// TwinCAT 3 PLC project PLCproj
// ProgramVersion: 3.1.4020.10
// libraries:
//   Tc2_Database, * (Beckhoff Automation GmbH)
//   Tc2_Standard, * (Beckhoff Automation GmbH)
//   Tc2_System, * (Beckhoff Automation GmbH)
//   Tc2_Utilities, * (Beckhoff Automation GmbH)
//   Tc3_Module, * (Beckhoff Automation GmbH)
//   VisuDialogs, * (System)
// project tree:
//   DUTs/ E_ACtype.TcDUT, E_Direction.TcDUT, E_Nchannel.TcDUT, ST_Terminal.TcDUT
//   / GlobalTextList.TcGTLO, PlcTask.TcTTO, Visualization Manager.TcVMO (not stored)
//   GVLs/ GVL.TcGVL, GVL_Checks.TcGVL
//   POUs/ FB_WriteReportToFile.TcPOU, F_Scaling.TcPOU, MAIN.TcPOU, P_Test.TcPOU
//   POUs/Checks/ CheckBounds.TcPOU, CheckDivDInt.TcPOU, CheckDivLInt.TcPOU, CheckDivLReal.TcPOU, CheckDivReal.TcPOU, CheckPointer.TcPOU, CheckRangeSigned.TcPOU, CheckRangeUnsigned.TcPOU
//   VISUs/ Screen1.TcVIS, Obrazki.TcIPO (not stored)
//   VISUs/TextList/ TL_ACtype.TcTLO, TL_BitConventer.TcTLO, TL_Busy.TcTLO, TL_Device.TcTLO, TL_Direction.TcTLO, TL_Nchannel.TcTLO
// real-time tasks:
//   TASK PlcTask: cycle T#10ms, priority 20, ADS port 350
// I/O:
//   DEVICE Device 2 (CX-BK)
//     Box 1 (CX-BK)
// variable links:
//   PLCproj/PLCproj Instance <-> Device 2 (CX-BK)/Box 1 (CX-BK)
//     PlcTask Inputs/GVL.aiINchannel[{1..4}] <-> Term 3 (KL3064)/Channel {1..4}/Data In  (4 links)
//     PlcTask Outputs/GVL.aiOUTchannel[{1..4}] <-> Term 2 (KL4404)/Channel {1..4}/Data Out  (4 links)

CONFIGURATION PLCproj
    RESOURCE PLC ON TwinCAT3
        TASK PlcTask(INTERVAL := T#10ms, PRIORITY := 20);
        PROGRAM MAIN WITH PlcTask : MAIN;
    END_RESOURCE
END_CONFIGURATION

// ---- DUTs/E_ACtype.TcDUT
TYPE E_ACtype :
(
	eACtype_null		:= 0,
	eACtype_0_10V		:= 1,
	eACtype_pl_min10V	:= 2,
	eACtype_0_20mA	:= 3,
	eACtype_4_20mA	:= 4
);
END_TYPE

// ---- DUTs/E_Direction.TcDUT
TYPE E_Direction :
(
	eDirection_null := 0,
	eDirection_Input_Module := 1,
	eDirection_Output_Module := 2
);
END_TYPE

// ---- DUTs/E_Nchannel.TcDUT
TYPE E_Nchannel :
(
	eNchannel_null := 0,
	eNchannel_2 := 1,
	eNchannel_4 := 2,
	eNchannel_8 := 3
);
END_TYPE

// ---- DUTs/ST_Terminal.TcDUT
TYPE ST_Terminal :
STRUCT
	usiDirection		:	USINT;							// Input=1  Output=2
	usiACtype			:	USINT;							// 0..10__±10V__0..20mA__4..20mA 
	usiNchannel			:	USINT;							// Amount of channel
	usiBitConventer		:	USINT;							// N-bit conventer
	sParameters			:	STRING(256);					// Message displayed in HMI during setup terminal type
END_STRUCT
END_TYPE

// ---- GVLs/GVL.TcGVL
VAR_GLOBAL
	 aiINchannel		AT %I*	:	ARRAY [1..8] OF  INT;
	 aiOUTchannel		AT %Q*	:	ARRAY [1..8] OF  INT;
	 

	 
	// aiINchannel		:	ARRAY [1..8] OF  INT;
	// aiOUTchannel		:	ARRAY [1..8] OF  INT;
END_VAR

// ---- GVLs/GVL_Checks.TcGVL
{attribute 'qualified_only'}
VAR_GLOBAL PERSISTENT
	dCheckBounds		: DINT;	(*Licznik przekroczen zakresu indexow, np. tablic*)
	dCheckDivDInt		: DINT;	(*Licznik prob dzielenia Dint przez 0*)
	dCheckDivLInt		: DINT; (*Licznik prob dzielenia LInt przez 0*)
	dCheckDivLReal		: DINT; (*Licznik prob dzielenia LREAL przez 0*)
	dCheckDivReal		: DINT; (*Licznik prob dzielenia REAL przez 0*)
	dCheckRangeSigned	: DINT;	(*Licznik przekroczen  liczby znakowej*)
	dCheckRangeUnsigned	: DINT; (*Licznik przekroczen  liczby bezznakowej*)
END_VAR

// ---- POUs/MAIN.TcPOU
(************************************************************************************)
(*							Beckhoff Automation Poland								*)
(*									13.09.2016										*)
(*								autor: Piotr Szyszka								*)
(*		Analog tester. Allows to chceck suspected with referenced terminal.			*)
(*						Please check preferences in local files.					*)
(*__________________________________________________________________________________*)
PROGRAM MAIN
VAR

END_VAR

P_Test();

END_PROGRAM

// ---- POUs/P_Test.TcPOU
(************************************************************************************)
(*							Beckhoff Automation Poland								*)
(*									13.09.2016										*)
(*								Analog terminal tester								*)
(*								autor: Piotr Szyszka								*)
(*																					*)
(*__________________________________________________________________________________*)
PROGRAM P_Test
VAR
// Choose bus terminals
bReadData			:	BOOL;							// Read Structure
bErrorReadData		:	BOOL;							// Setted not all parametres
bDataSend			:	BOOL;							// Data aquired
stRefTerminal		:	ST_Terminal;
stTestTerminal		:	ST_Terminal;
rtReadData			:	R_TRIG;
ftClearComboBox		:	F_TRIG;
sStatusBox			:	STRING(255)		:='Idle';
sBuffer				:	STRING(255);

eDirection1			:	E_Direction;					// Input=1  Output=2
eDirection2			:	E_Direction;
eACtype				:	E_ACtype;						// 0..10V=1	±10V=2	0..20mA=3	4..20mA=4
eNchannel			:	E_Nchannel;						// 2channels=2	4channels=4		8channels=8

// Test
bTestEnable				:	BOOL;					// Launch Test procedure
bTestBusy				:	BOOL;					// Test- busy marker: 1-runned_procedure 0-stopped_procedure
usiTestCycle			:	USINT	:=	3;			// Amount of test cycle
iStep					:	INT		:=	0;			// Actual procedure function
usiActualChannelNumber	:	USINT;					// Actual tested channel
usiActualCycle			:	USINT;					// Actual test cycle 
uiFullfilment			:	UINT;					// Percent of signal fullfilment
usiProcedure			:	USINT;					// Actual procedure
rPercent				:	REAL;					// TestValue/RefValue [%]
usiOKsamples			:	USINT;					// Variable summing positive test results.
usiERRORsamples			:	USINT;					// Variable summing negative test results.

// fbGetTime
fbGetTime				:	NT_GetTime;
tpPulse					:	TP;
rtPulse					:	R_TRIG;

// fbWriteReportToFile
fbWriteReportToFile		:	FB_WriteReportToFile;	
rtTestEnable			:	R_TRIG;					// Detecting entering procedure
ftBreakProcedure		:	F_TRIG;					// Detecting user terminating procedure 
rtWriteReportToFile		:	R_TRIG;					// Detecting start of saving
ftWriteReportToFile		:	F_TRIG;					// Detecting end of saving
stActTime				:	TIMESTRUCT;
sData					:	STRING(255);			// Variables transfered to actual row in raport
sPath					:	STRING(255);
usiTestNumber			:	USINT;
bWrite					:	BOOL;					// Send data on demand
tonWait					:	TON;					// Works like 'Continue' in C language
tpWait					:	TP;						// Works like 'Continue' in C language

// f_Scalling
rXmin					:	REAL;
rXmax					:	REAL;
rYmin					:	REAL;
rYmax					:	REAL;
END_VAR

A_ChooseBusTerminals();		// Action Block- Visualisation

tpPulse(IN:= NOT tpPulse.Q, PT:= T#1S);
rtPulse(CLK:= tpPulse.Q);
fbGetTime(	START:= rtPulse.Q,
			TMOUT:= T#2S,
			TIMESTR=> stActTime);

rtWriteReportToFile(clk:=bWrite);
ftWriteReportToFile();
fbWriteReportToFile(sHeader:='Czas$tFullfilment [%]$tActChannel$tActCycle$tTestTerminalValue [INT]$tRefTerminalValue [INT]$tTestTerminalValue [V / mA]$tRefTerminalValue [V / mA]$tTestValue/RefValue [%]$tStatus$n',	
					sData:= sData,
					sPath:= sPath,
					stActTime:= stActTime,
					wNewFileFrequency:= 0,
					bWrite:= rtWriteReportToFile.Q,		// Write od demand
					bBusy=> ftWriteReportToFile.CLK );
					
tonWait(PT:=T#15MS);	// timer- Works like 'Continue' in C language

CASE iStep OF
0:	// Detecting start procedure
	rtTestEnable(clk:=bTestEnable);
	IF(rtTestEnable.Q AND bErrorReadData=FALSE)	THEN	
		usiTestNumber:= usiTestNumber + 1;
		sBuffer:= USINT_TO_STRING(usiTestNumber);
		sPath:=	CONCAT('C:\Users\Administrator\Desktop\Raport',sBuffer);	// set next file name
		sPath:=	CONCAT(sPath,'_');
	
		bTestBusy:=TRUE;
		iStep:=10;
	END_IF
	
10:	// Initialization
	usiActualChannelNumber:= 1; 		
	usiActualCycle:= 1;
	uiFullfilment:= 0;
	bWrite:= FALSE;
	usiOKsamples:= 0;
	usiERRORsamples:= 0;
	
	CASE stTestTerminal.usiACtype OF	// Choosing right procedure
		1:	usiProcedure:=1;	// Procedure 1:		Analog > Analog		12-bit		0..10V
		2:	usiProcedure:=2;	// Procedure 2:		Analog > Analog		12-bit		-10V .. +10V
		3:	usiProcedure:=3;	// Procedure 3:		Analog > Analog		12-bit		0..20mA
		4:	usiProcedure:=4;	// Procedure 4:		Analog > Analog		12-bit		4..20mA
	END_CASE
	iStep:= 20;
						
20:	// Sending header of report procedure to file
	CASE usiProcedure OF	// Choosing right procedure
		1:	sData:= 'STARTING PROCEDURE 1: ANALOG > ANALOG 12-bit 0..10V (0..0X7FFF)$n';
		2:	sData:= 'STARTING PROCEDURE 2: ANALOG > ANALOG 12-bit -10V..+10V (0x8000..0X7FFF)$n';
		3:	sData:= 'STARTING PROCEDURE 3: ANALOG > ANALOG 12-bit 0..20mA (0..0X7FFF)$n';
		4:	sData:= 'STARTING PROCEDURE 4: ANALOG > ANALOG 12-bit 4..20mA (0..0X7FFF)$n';
	END_CASE
	
	bWrite:= TRUE;	// Send data to XLS raport. Wait for save.
	IF(ftWriteReportToFile.Q)	THEN	
		bWrite:=FALSE;
		iStep:= 21;
	END_IF
	
21:	sData:='_______________________________________________________________________________________$n';
	
	bWrite:= TRUE;	// Send data to XLS raport. Wait for save.
	IF(ftWriteReportToFile.Q)	THEN	
		bWrite:=FALSE;
		iStep:= 30;
	END_IF
	
30:	// Testing channel by channel. 
	IF(usiActualChannelNumber<=stTestTerminal.usiNchannel)	THEN
		iStep:= 40;
	ELSE
		// Properly end of procedure raport 
		sBuffer:= 'Test Completed!$n$tSummary:$n$t$tNumber of "OK" results:$t';
		sData:= CONCAT(sBuffer,USINT_TO_STRING(usiOKsamples));
		
		sBuffer:= '$n$t$tNumber of "ERROR" samples:$t';	
		sData:= CONCAT(sData,sBuffer);	
		sData:= CONCAT(sData,USINT_TO_STRING(usiERRORsamples));
		
		bWrite:= TRUE;	// Send data to XLS raport. Wait for save.
		IF(ftWriteReportToFile.Q)	THEN	
			bWrite:=FALSE;
			iStep:= 70;
		END_IF
	END_IF
	
40:	// Checking amount of cycles
	IF(usiActualCycle<=usiTestCycle) THEN // test 0..100% Volt fullfilment 
		iStep:= 50;
	ELSE	// test next channel
		usiActualChannelNumber:= usiActualChannelNumber+1;
		usiActualCycle:= 1;
		iStep:= 30; // Check again ActualChannel
	END_IF
	
50:	// Increasing Voltage
	CASE usiProcedure OF
		1:	rXmin:=	0;	rXmax:= 100;	rYmin:= 0;		rYmax:= 32767;
		2:	rXmin:=	0;	rXmax:= 100;	rYmin:= -32768;	rYmax:= 32767;
		3:	rXmin:=	0;	rXmax:= 100;	rYmin:= 0;		rYmax:= 32767;
		4:	rXmin:=	0;	rXmax:= 100;	rYmin:= 0;		rYmax:= 32767;
	END_CASE
	IF(uiFullfilment<100)	THEN
		IF (uiFullfilment=0)	THEN
			aiOUTchannel[usiActualChannelNumber]:= REAL_TO_INT(	F_Scaling(	rValue:= uiFullfilment,
																		rXmin:= rXmin, rXmax:= rXmax,
																		rYmin:= rYmin, rYmax:= rYmax));
			uiFullfilment:=uiFullfilment+1;
		ELSE
			uiFullfilment:=uiFullfilment+1;
			aiOUTchannel[usiActualChannelNumber]:= REAL_TO_INT(	F_Scaling(	rValue:= uiFullfilment,
																		rXmin:= rXmin, rXmax:= rXmax,
																		rYmin:= rYmin, rYmax:= rYmax));
		END_IF
	ELSE
		usiActualCycle:= usiActualCycle+1;
		uiFullfilment:= 0;
		iStep:= 40;
		RETURN;		// 'Continue'
	END_IF
	iStep:= 60;
	
60:	// Actual probe raport
	tonWait.IN := TRUE;	// Wait for next PLC cycle for gain I/O data.
	IF tonWait.Q THEN
		CASE usiProcedure OF	// INT to Volt/mAmper scalling
			1:	rXmin:=	0;		rXmax:= 32767;	rYmin:= 0;		rYmax:= 10;
			2:	rXmin:=	-32768;	rXmax:= 32767;	rYmin:= -10;	rYmax:= 10;
			3:	rXmin:=	0;		rXmax:= 32767;	rYmin:= 0;		rYmax:= 20;
			4:	rXmin:=	0;		rXmax:= 32767;	rYmin:= 4;		rYmax:= 20;
		END_CASE
		
		sData:= UINT_TO_STRING(uiFullfilment);
		sData:= CONCAT(sData, '$t');	
		
		sBuffer:=USINT_TO_STRING(usiActualChannelNumber);
		sData:= CONCAT(sData, sBuffer);
		sData:= CONCAT(sData, '$t');
		
		sBuffer:=USINT_TO_STRING(usiActualCycle);
		sData:= CONCAT(sData, sBuffer);
		sData:= CONCAT(sData, '$t');
		
		sBuffer:=INT_TO_STRING( aiINchannel[usiActualChannelNumber] );
		sData:= CONCAT(sData, sBuffer);
		sData:= CONCAT(sData, '$t');
		
		sBuffer:=INT_TO_STRING( aiOUTchannel[usiActualChannelNumber] );
		sData:= CONCAT(sData, sBuffer);
		sData:= CONCAT(sData, '$t');	
		
		sBuffer:=REAL_TO_STRING(	F_Scaling(	rValue:= aiINchannel[usiActualChannelNumber],
												rXmin:= rXmin, rXmax:= rXmax,
												rYmin:= rYmin, rYmax:= rYmax)	);
		sData:= CONCAT(sData, sBuffer);
		sData:= CONCAT(sData, '$t');	
		
		sBuffer:=REAL_TO_STRING(	F_Scaling(	rValue:= aiOUTchannel[usiActualChannelNumber],
												rXmin:= rXmin, rXmax:= rXmax,
												rYmin:= rYmin, rYmax:= rYmax)	);
		sData:= CONCAT(sData, sBuffer);
		sData:= CONCAT(sData, '$t');
		
		IF(aiOUTchannel[usiActualChannelNumber]=0)	THEN
			sBuffer:='DIV/0 !'; // Division by 0!
		ELSE
			rPercent:= INT_TO_REAL(aiINchannel[usiActualChannelNumber]) / INT_TO_REAL(aiOUTchannel[usiActualChannelNumber]) *100;
			sBuffer:=REAL_TO_STRING(rPercent);
		END_IF
		sData:= CONCAT(sData, sBuffer);
		sData:= CONCAT(sData, '$t');	
		
		IF(aiOUTchannel[usiActualChannelNumber]<>0 AND rPercent>95 AND rPercent<105)	THEN	// Set error limit (default 95..105% is OK)
			sBuffer:='OK';
			usiOKsamples:= usiOKsamples+1;
		ELSIF(aiOUTchannel[usiActualChannelNumber]=0)	THEN
			sBuffer:='null'; // Division by 0!
		ELSE
			sBuffer:='ERROR';
			usiERRORsamples:= usiERRORsamples+1;
		END_IF
		sData:= CONCAT(sData, sBuffer);
		sData:= CONCAT(sData, '$n');	// endl. Ready to send
		
		IF(uiFullfilment=100 AND usiActualCycle=usiTestCycle)	THEN
			sBuffer:= '$t-$tNext channel$n';
			sData:= CONCAT(sData, sBuffer);
		ELSIF(uiFullfilment=100)	THEN	// Additional text for next cycle, channel...
			sBuffer:= '$t-$t$tNext cycle$n';
			sData:= CONCAT(sData, sBuffer);
		END_IF
		
		bWrite:= TRUE;
	END_IF	
	IF(ftWriteReportToFile.Q)	THEN
		bWrite:=FALSE;
		tonWait.IN := FALSE;
		iStep:= 65;
	END_IF

65:	// Refresh sStatusBox in VISU
	sStatusBox:= 'Raport file path:$n';
	sStatusBox:= CONCAT(sStatusBox, sPath);
	
	sBuffer:= '$nActual Status:$nFullfilment: ';
	sStatusBox:= CONCAT(sStatusBox, sBuffer);
	
	sBuffer:= UINT_TO_STRING(uiFullfilment);
	sStatusBox:= CONCAT(sStatusBox, sBuffer);
	
	sBuffer:= '% | Actual Cycle: ';
	sStatusBox:= CONCAT(sStatusBox, sBuffer);
	
	sBuffer:= USINT_TO_STRING(usiActualCycle);
	sStatusBox:= CONCAT(sStatusBox, sBuffer);
	
	sBuffer:= ' | Actual Channel: ';
	sStatusBox:= CONCAT(sStatusBox, sBuffer);
	
	sBuffer:= USINT_TO_STRING(usiActualChannelNumber);
	sStatusBox:= CONCAT(sStatusBox, sBuffer);
	
	iStep:= 80;
	
70:	// Quit procedure
	IF(sStatusBox<>'Procedure terminated by user!')	THEN	
		sStatusBox:= 'Test completed!$nNumber of ERROR samples: ';	
		sStatusBox:= CONCAT(sStatusBox,USINT_TO_STRING(usiERRORsamples));
		IF(usiERRORsamples=0)	THEN
			sStatusBox:= CONCAT(sStatusBox,'$nTested terminal works correctly.');
		END_IF
	END_IF
	bTestBusy:=FALSE;
	iStep:=0;

80: // Detecting break procedure- Terminated by user
	ftBreakProcedure(CLK:= bTestEnable);
	IF(ftBreakProcedure.Q = TRUE) THEN
		sData:= 'Procedure terminated by user!$n';
		sStatusBox:= 'Procedure terminated by user!';
		bWrite:= TRUE;
	ELSIF(ftWriteReportToFile.Q AND bTestEnable=FALSE)	THEN	// wait for write
			bWrite:=FALSE;
			iStep:= 70;
	ELSIF (bWrite=FALSE)	THEN
		iStep:= 50;	// go back to procedure
	END_IF
	
END_CASE

ACTION A_ChooseBusTerminals:
rtReadData(clk:= bReadData);

// Loading terminals parameters from HMI
IF(rtReadData.Q)	THEN
	IF(	eDirection1>0 AND eDirection2>0 AND eACtype>0 AND eNchannel>0) THEN // chceck if all fields in HMI was choosen properly
			// Tested terminal
			stTestTerminal.usiDirection:= INT_TO_USINT(eDirection1);
			stTestTerminal.usiACtype:= INT_TO_USINT(eACtype);
			CASE eNchannel OF
				1:	stTestTerminal.usiNchannel:= 2;
				2:	stTestTerminal.usiNchannel:= 4;
				ELSE stTestTerminal.usiNchannel:= 8;
			END_CASE	
			
			// Reference terminal
			stRefTerminal.usiDirection:= INT_TO_USINT(eDirection2);
			
			bErrorReadData:= FALSE;
			bDataSend:= TRUE;
			sStatusBox:= 'Data Aquired';
		
	ELSE // error input data
			bErrorReadData:= TRUE;
			bDataSend:= FALSE;
			sStatusBox:= 'Not enough input arguments!';
	END_IF	
END_IF


// Zerowanie Combo Box w HMI
ftClearComboBox(clk:= bDataSend);
IF( ftClearComboBox.Q AND ( LEN(stRefTerminal.sParameters)>30 OR LEN(stTestTerminal.sParameters)>30 ) )	THEN
	eDirection1:=0;
	eACtype:=0;
	eNchannel:=0;
	eDirection2:=0;
END_IF
END_ACTION

END_PROGRAM

// ---- POUs/FB_WriteReportToFile.TcPOU
(****************************************************************************************************)
(*							Beckhoff Automation Poland												*)
(*							FB_WriteReportToFile v1.5												*)
(*					v1.2 - internal optimizations													*)
(*					v1.3 - internal optimizations													*)
(*					v1.4 - zmiana funkcjonalności, obsługa błędów, większa elastyczność				*)
(*					v1.5 - dodanie bufora zapisu, poprawienie zapisu Header							*)
(*									06.06.2012														*)
(*				Blok funkcyjny slużący do zapisywania danych do pliku *.xls.						*)
(*					Pierwszy wiersz kazdego pliku stanowi sHeader.									*)
(*	Zapisywane sData, podawane są na wejście bloku funkcyjnego jako zmienna typu STRING.			*)
(*				Pierwsza kolumna zawiera datę i godzinę wykonania wpisu.							*)
(*				Możliwe jest ustawienie częstości zapisywania do pliku,								*)
(* 			Konieczne jest dodanie biblioteki TcUtilities.lib, TcSystem.lib oraz TcBase.lib			*)
(*		UWAGA!!!																					*)
(*		Blok ten korzysta z czasu systemowego, podawanego na wejście bloku.							*)
(*		Nie można wywoływać tego bloku bez podania czasu na wejściu,								*)
(*		ponieważ wówczas przyjmuje on wartości zerowe i blok nie wykona zapisu						*)
(*		BLOK FUNKCYJNY DZIAŁA TYLKO DLA "PC OR CX( x86)"											*)
(*__________________________________________________________________________________________________*)

FUNCTION_BLOCK FB_WriteReportToFile
VAR_INPUT
	sHeader:				STRING(255);(*:='Czas$tKolumna1$tKolumna2$tKolumna3$n';*)	(* Naglowki kolumn - cała górna linia - powinna być zakończona '$n'*)
 	sData: 					STRING(255);(*:='Zmienna1$tZmienna2$tZmienna3$n'; *)		(* sData do zapisu w postaci napisu, np 'test$n', 10 znaków zajmie stempel czasowy z przodu - dołączony zostanie automatycznie, więc max długość linii 245 znaków!!!!!! *)
	sPath:					STRING(255);(*:='c:\';*)									(* sPath zapisu pliku bez nazwy pliku, np 'c:\' *)
	stActTime:				TIMESTRUCT;													(* Aktualny czas w formie struktury - TIMESTRUCT *)
	tWriteFrequency:		TIME; 												(* Częstotliwość zapisu do pliku *)
	wNewFileFrequency:		WORD:=0;													(* Częstotliwość tworzenia nowego pliku: dzien (0), tydzien(1), miesiac(2) *)
	bWrite: 				BOOL; 														(* Zapis na rozkaz *)
END_VAR
VAR_OUTPUT
	bBusy: 					BOOL;		(* Sygnał zajętości bloczka *)
	bError:					BOOL;		(* Flaga błedu, bloczek sam się resetuje, więc flaga mnoże samoczynnie zniknąć *)
	dwErrors:				DWORD;		(* Suma błędów od uruchomienia programu PLC *)
	dwErrorsInCurrentFile:	DWORD;		(* Suma błedów zapisu do nowego pliku lub od uruchomienia *)
END_VAR

VAR
	sFileName: 				STRING;
	fbFileOpen: 			FB_FileOpen;
	fbFileWrite:  			FB_FilePuts;
	fbFileClose: 			FB_FileClose;
	Step: 					INT;
	TrigerName:				R_TRIG;
	sTime: 					STRING(10);										(*odciecie min rozmiarem*)
	sTimeExcel: 			STRING(19);										(*odciecie min rozmiarem*)
	stActTimeName:			TIMESTRUCT;										(* Aktualny czas w formie struktury użyty do tworzenia nazwy pliku *)
	sOldName:				STRING:='start';
	bInitialization: 		BOOL:=TRUE;
	WriteTimer: 			TON;
	WatchDog:				TON;
	rtWrite: 				R_TRIG; 										(* 1-krotny zapis na zadanie *)
	fbBuffer:				FB_StringRingBuffer;							(*Bufor zapisu*)
	arrBuffer: 				ARRAY [1..20] OF STRING(255);					(*Tablica bufora zapisu*)
	sLine:					STRING(255);									(*Linia do zapisu*)
END_VAR

(* Akcja wywołująca bloki w tle *)
CallBackgroundFBs();
(*Akcja Name*)
Name();
(*Obsługa bufora zapisu*)
fbBuffer(pBuffer:= ADR(arrBuffer),
		cbBuffer:= SIZEOF(arrBuffer));
(*Dodawanie elementów do bufora*)
IF rtWrite.Q THEN
	fbBuffer.A_AddTail(putValue:= sData);
END_IF
CASE Step OF
	0: (* Initialization *)
		IF stActTime.wYear<>0 THEN
			(*format daty  w pliku Excela*)
			sTimeExcel:=SYSTEMTIME_TO_STRING(stActTime);
			WatchDog.IN:= TRUE;
			fbFileOpen.bExecute:= TRUE;
			bBusy := TRUE;
			bError := FALSE;
			bInitialization:=FALSE;
			fbFileOpen.bExecute := TRUE;
			fbFileOpen.nMode := FOPEN_MODEREAD;
			Step:= Step+5;
		END_IF
	5:	(*Sprawdzenie czy plik jest stworzony*)
		IF fbFileOpen.bBusy = FALSE AND NOT fbFileOpen.bError THEN
			Step := 60;
			sOldName := sFileName;
			fbFileOpen.bExecute := FALSE;
			fbFileClose.bExecute:= TRUE;
			fbFileOpen.nMode:= FOPEN_MODEAPPEND OR FOPEN_MODEPLUS ;
		ELSIF fbFileOpen.bError THEN
			Step := 20;
			fbFileOpen.bExecute := FALSE;
			fbFileOpen.nMode:= FOPEN_MODEAPPEND OR FOPEN_MODEPLUS ;
		END_IF
	10: (* Waiting for write request *)
		fbBuffer.A_RemoveHead(getValue=> sLine);
		IF fbBuffer.bOk AND sLine <> '' THEN
			(*format daty  w pliku Excela*)
			sTimeExcel:=SYSTEMTIME_TO_STRING(stActTime);
			WatchDog.IN:= TRUE;
			fbFileOpen.bExecute:= TRUE;
			bBusy := TRUE;
			bError := FALSE;
			Step := Step + 10;
		END_IF

	20:	(*Otwieramy plik*)
		fbFileOpen.bExecute := TRUE;
		IF fbFileOpen.bBusy = FALSE AND NOT fbFileOpen.bError THEN
			fbFileOpen.bExecute:= FALSE;
		(*Tworzene nowego pliku z naglowkiem*)
			IF sOldName = sFileName THEN
				(*do istniejacego pliku dopisujemy sData*)
				Step := Step + 20;
			ELSE
				(* Kasujemy błedy bieżącego pliku *)
				dwErrorsInCurrentFile := 0;
				(*Wysylamy sHeader*)
				fbFileWrite.bExecute:= TRUE;
				fbFileWrite.sLine := sHeader;
				sOldName := sFileName;
				Step := Step + 10;
			END_IF
		END_IF

	30:
		IF fbFileWrite.bBusy = FALSE AND NOT fbFileWrite.bError THEN
			fbFileWrite.bExecute:= FALSE;
			Step :=  50;
		END_IF

	40:	(*Wysylamy sLine*)
		fbFileWrite.bExecute:= TRUE;
		sTimeExcel := DELETE (sTimeExcel,1,11);(*usuniecie znaku' -' przed godzina*)
		sTimeExcel := INSERT (sTimeExcel,' ',10);(*wstawienie znaku ' ' przed godzina *)

		sLine:=CONCAT('$t',sLine);
		sLine:=CONCAT(sTimeExcel,sLine);
		fbFileWrite.sLine := sLine;
		Step := Step + 10;
	50:
		IF fbFileWrite.bBusy = FALSE AND NOT fbFileWrite.bError THEN
			fbFileWrite.bExecute:= FALSE;
			fbFileClose.bExecute:= TRUE;
			Step := Step + 10;
		END_IF

	60:	(*Zamykanie pliku*)
		IF fbFileClose.bBusy = FALSE AND fbFileClose.bError = FALSE THEN
			fbFileClose.bExecute:= FALSE;
			bBusy := FALSE;
			WatchDog.IN:= FALSE;
			Step := 10;
		END_IF
	99: (* Error *)
		fbFileOpen.bExecute:= FALSE;
		fbFileWrite.bExecute:= FALSE;
		fbFileClose.bExecute:= FALSE;
		WatchDog.IN:= FALSE;
		bError := TRUE;
		dwErrors := dwErrors + 1;
		dwErrorsInCurrentFile := dwErrorsInCurrentFile + 1;
		Step := 10;
END_CASE
CallFileFBs();

ACTION CallBackgroundFBs:
(*Wywolanie blokow funkcyjnych*)
TrigerName();
rtWrite(CLK:= bWrite);

(*Reset bloczka w przypadku bledu*)
WatchDog(PT:=T#10s);
IF WatchDog.Q THEN  Step:=99; END_IF

(*Ustalenie czestotliwosci zapisu do pliku*)
WriteTimer(IN:= NOT WriteTimer.Q, PT:= tWriteFrequency, Q=> , ET=> );
END_ACTION

ACTION CallFileFBs:
(*Wywołanie bloków odpowiedzialnych za zapisywanie*)
fbFileOpen(
	sNetId:= '',
	sPathName:= sFileName,
	ePath:= PATH_GENERIC,
	tTimeout:= T#200ms);

fbFileWrite(
	sNetId:= '',
	hFile:= fbFileOpen.hFile,
	tTimeout:= T#250ms);

fbFileClose(
	sNetId:= '',
	hFile:= fbFileOpen.hFile,
	tTimeout:= t#200ms);
END_ACTION

ACTION Name:
(*xxxxxxxxxxxxxxxxxxxxxxxxxxxxxxxxxxxxxxxxxxxxxxxxxxxxxxxxxxxxxxxxxxxxxxxxxxxxxxxxxxxxxxxxxxxxxxxxxxxxxxxxxxxxxxxx
				Ustalenie częstotliwości twrzenia nowego pliku i zmiana nazwy pliku
xxxxxxxxxxxxxxxxxxxxxxxxxxxxxxxxxxxxxxxxxxxxxxxxxxxxxxxxxxxxxxxxxxxxxxxxxxxxxxxxxxxxxxxxxxxxxxxxxxxxxxxxxxxxxxxxx*)
CASE wNewFileFrequency OF
	0:	(*Tworzenie pliku raz dziennie*)
		stActTimeName := stActTime;
		stActTimeName.wHour := 0;
		stActTimeName.wMinute := 0;

	1:	(*Tworzenie pliku raz w tygodniu*)
		IF bInitialization THEN
			stActTimeName := stActTime;
			stActTimeName.wHour := 0;
			stActTimeName.wMinute := 0;
		ELSIF stActTime.wDayOfWeek = 1 THEN
			stActTimeName := stActTime;
			stActTimeName.wHour := 0;
			stActTimeName.wMinute := 0;
		END_IF
ELSE
		(*Tworzenie pliku raz w miesiącu*)
		stActTimeName := stActTime;
		stActTimeName.wDay := 1;
		stActTimeName.wHour := 0;
		stActTimeName.wMinute := 0;

END_CASE

sTime := SYSTEMTIME_TO_STRING(stActTimeName);
sTime := DELETE (sTime,1,11);(*usuniecie znaku' -' przed godzina*)
sFileName:=CONCAT(sPath,sTime);
sFileName:=CONCAT(sFileName,'.xls');
END_ACTION

END_FUNCTION_BLOCK

// ---- POUs/F_Scaling.TcPOU
(************************************************************************************)
(*							Beckhoff Automation Poland								*)
(*								F_Scaling v2										*)
(*									3.11.2011										*)
(*					Funkcja skalująca wartość wejściową rValue na wyjściową 		*)
(*__________________________________________________________________________________*)
FUNCTION F_Scaling: REAL
VAR_INPUT
	rValue	:	REAL;	(*Zmienna skalowana*)
	rXmin	:	REAL;	(*Dolny zakres zmiennej przeskalowanej*)
	rXmax	:	REAL;	(*Górny zakres zmiennej przeskalowanej*)
	rYmin	:	REAL;	(*Dolny zakres zmiennej skalowanej*)
	rYmax	:	REAL;	(*Górny zakres zmiennej skalowanej*)
END_VAR
VAR
	rfA		:	REAL;	(*Wspólczynnik kierunkowy prostej*)
	rfB		:	REAL;	(*Współczynnik przesunięcia prostej*)
END_VAR

IF (rValue > rXmax) THEN
	F_Scaling := rYmax;
ELSIF (rValue <= rXmin) THEN
	F_Scaling := rYmin;
ELSE
	IF (((rXmax - rXmin) < 0.01) AND ((rXmax - rXmin) > -0.01)) THEN
		F_Scaling := rYmin;
	ELSE
		rfA := (rYmax - rYmin) / (rXmax - rXmin);
		rfB := rYmax - rfA * rXmax;
		F_Scaling := rfA * rValue + rfB;
	END_IF;
END_IF

END_FUNCTION

// ---- POUs/Checks/CheckBounds.TcPOU
// Implicitly generated code : DO NOT EDIT
FUNCTION CheckBounds : DINT
VAR_INPUT
	index, lower, upper: DINT;
END_VAR

// Implicitly generated code : Only an Implementation suggestion
IF  index < lower THEN
	CheckBounds := lower;
	GVL_Checks.dCheckBounds := GVL_Checks.dCheckBounds + 1;
ELSIF  index > upper THEN
	CheckBounds := upper;
	GVL_Checks.dCheckBounds := GVL_Checks.dCheckBounds + 1;
ELSE  
	CheckBounds := index;
END_IF

END_FUNCTION

// ---- POUs/Checks/CheckDivDInt.TcPOU
// Implicitly generated code : DO NOT EDIT
FUNCTION CheckDivDInt : DINT
VAR_INPUT
	divisor:DINT;
END_VAR

// Implicitly generated code : Only an Implementation suggestion
IF divisor = 0 THEN
	CheckDivDInt:=1;
	GVL_Checks.dCheckDivDInt := GVL_Checks.dCheckDivDInt + 1;
ELSE
	CheckDivDInt:=divisor;
END_IF;

END_FUNCTION

// ---- POUs/Checks/CheckDivLInt.TcPOU
// Implicitly generated code : DO NOT EDIT
FUNCTION CheckDivLInt : LINT
VAR_INPUT
	divisor:LINT;
END_VAR

// Implicitly generated code : Only an Implementation suggestion
IF divisor = 0 THEN
	CheckDivLInt:=1;
	GVL_Checks.dCheckDivLInt := GVL_Checks.dCheckDivLInt + 1;
ELSE
	CheckDivLInt:=divisor;
END_IF;

END_FUNCTION

// ---- POUs/Checks/CheckDivLReal.TcPOU
// Implicitly generated code : DO NOT EDIT
FUNCTION CheckDivLReal : LREAL
VAR_INPUT
	divisor:LREAL;
END_VAR

// Implicitly generated code : Only an Implementation suggestion
IF divisor = 0 THEN
	CheckDivLReal:=1;
	GVL_Checks.dCheckDivLReal := GVL_Checks.dCheckDivLReal + 1;
ELSE
	CheckDivLReal:=divisor;
END_IF;

END_FUNCTION

// ---- POUs/Checks/CheckDivReal.TcPOU
// Implicitly generated code : DO NOT EDIT
FUNCTION CheckDivReal : REAL
VAR_INPUT
	divisor:REAL;
END_VAR

// Implicitly generated code : Only an Implementation suggestion
IF divisor = 0 THEN
	CheckDivReal:=1;
	GVL_Checks.dCheckDivReal := GVL_Checks.dCheckDivReal + 1;
ELSE
	CheckDivReal:=divisor;
END_IF;

END_FUNCTION

// ---- POUs/Checks/CheckPointer.TcPOU
// Implicitly generated code : DO NOT EDIT
FUNCTION CheckPointer : POINTER TO BYTE
VAR_INPUT 
	ptToTest : POINTER TO BYTE; // Destination address of the pointer
	iSize : DINT;		        // Size of the type the pointer points to. (e.g: 20 for POINTER TO ARRAY [0..9] OF INT) 
	iGran : DINT;		        // Granularity of the pointer access. This is the size of the biggest non-structured data type in the type the pointer points to. (e.g: 2 for POINTER TO ARRAY [0..9] OF INT)
	bWrite: BOOL;		        // Indicates read or write Access. TRUE = write access.
END_VAR

// No standard way of implementation. Fill your own code here
CheckPointer := ptToTest;

END_FUNCTION

// ---- POUs/Checks/CheckRangeSigned.TcPOU
// Implicitly generated code : DO NOT EDIT
FUNCTION CheckRangeSigned : DINT
VAR_INPUT
	value, lower, upper: DINT;
END_VAR

// Implicitly generated code : Only an Implementation suggestion
IF (value < lower) THEN
	CheckRangeSigned := lower;
	GVL_Checks.dCheckRangeSigned := GVL_Checks.dCheckRangeSigned + 1;
ELSIF(value > upper) THEN
	CheckRangeSigned := upper;
	GVL_Checks.dCheckRangeSigned := GVL_Checks.dCheckRangeSigned + 1;
ELSE
	CheckRangeSigned := value;
END_IF

END_FUNCTION

// ---- POUs/Checks/CheckRangeUnsigned.TcPOU
// Implicitly generated code : DO NOT EDIT
FUNCTION CheckRangeUnsigned : UDINT
VAR_INPUT
	value, lower, upper: UDINT;
END_VAR

// Implicitly generated code : Only an Implementation suggestion
IF (value < lower) THEN
	CheckRangeUnsigned := lower;
	GVL_Checks.dCheckRangeUnsigned := GVL_Checks.dCheckRangeUnsigned + 1;
ELSIF(value > upper) THEN
	CheckRangeUnsigned := upper;
	GVL_Checks.dCheckRangeUnsigned := GVL_Checks.dCheckRangeUnsigned + 1;
ELSE
	CheckRangeUnsigned := value;
END_IF

END_FUNCTION

// ---- GlobalTextList.TcGTLO
TEXTLIST GlobalTextList
  12 = '%s'
  0 = 'Analog terminal tester'
  3 = 'Change'
  15 = 'Choose amount of channels'
  2 = 'Choose amount of test cycles per 1 channel'
  11 = 'Choose conventer precisions'
  1 = 'Choose module type'
  7 = 'Choose signals direction'
  10 = 'Choose signals range'
  8 = 'Choose type of module'
  9 = 'Choose type signals power'
  19 = 'Reference Device'
  4 = 'Run Test'
  6 = 'Send data to PLC'
  17 = 'START / STOP TEST'
  5 = 'Stop Test'
  18 = 'Tested Device'
  13 = 'Tested Device:\nModule type: \nSignals direction: \nType of module:\nType of signals power:\nSignals range:\nConventer precision:'
  14 = 'Tested Device:\nModule type: %s\nSignals direction: %s\nType of module: %s\nType of signals power: %s\nSignals range: %s\nConventer precision: %s'
  16 = 'TL_bBusy'
END_TEXTLIST

// ---- VISUs/Screen1.TcVIS
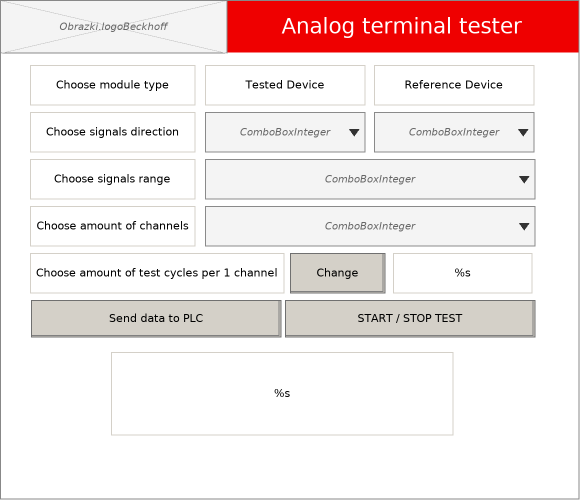
VISUALIZATION Screen1  // 580x500
    Rectangle (225,0 354x52), "Analog terminal tester"
    Image (0,0 227x53), image: Obrazki.logoBeckhoff
    Textfield (30,65 165x40), "Choose module type"
    Textfield (30,253 254x40), "Choose amount of test cycles per 1 channel"
    Button (285,300 250x37), "START / STOP TEST", colour toggle: P_Test.bTestBusy, pressed state: P_Test.bTestBusy
        p573394764: 16#FFFFFF00
        toggle P_Test.bTestEnable
    Button (31,300 250x37), "Send data to PLC", text variable: P_Test.bReadData, colour toggle: P_Test.bErrorReadData
        p573394764: 16#FFFF0000
        tap P_Test.bReadData
    Textfield (30,112 165x40), "Choose signals direction"
    Textfield (30,159 165x40), "Choose signals range"
    Textfield (393,253 139x40), "%s", text variable: P_Test.usiTestCycle
    Textfield (30,206 165x40), "Choose amount of channels"
    Button (290,253 95x40), "Change"
        OnMouseClick: write P_Test.usiTestCycle via VisuDialogs.Numpad, min 1, max 255
    ComboBoxInteger (205,112 160x40), variable: P_Test.eDirection1, text list: 'TL_Direction'
    ComboBoxInteger (205,159 330x40), variable: P_Test.eACtype, text list: 'TL_ACtype'
    ComboBoxInteger (205,206 330x40), variable: P_Test.eNchannel, text list: 'TL_Nchannel'
    Textfield (205,65 160x40), "Tested Device"
    ComboBoxInteger (374,112 160x40), variable: P_Test.eDirection2, text list: 'TL_Direction'
    Textfield (374,65 160x40), "Reference Device"
    Textfield (111,352 342x83), "%s", text variable: P_Test.sStatusBox
END_VISUALIZATION

// ---- VISUs/TextList/TL_ACtype.TcTLO
TEXTLIST TL_ACtype
  0 = 'Choose'
  1 = '0..10V'
  2 = '±10V'
  3 = '0..20mA'
  4 = '4..20mA'
   = ''
END_TEXTLIST

// ---- VISUs/TextList/TL_BitConventer.TcTLO
TEXTLIST TL_BitConventer
  0 = 'Choose'
  1 = '12-bit'
  2 = '16-bit'
   = ''
END_TEXTLIST

// ---- VISUs/TextList/TL_Busy.TcTLO
TEXTLIST TL_Busy
  0 = 'Begin Test'
  1 = 'Break Test'
   = ''
END_TEXTLIST

// ---- VISUs/TextList/TL_Device.TcTLO
TEXTLIST TL_Device
  0 = 'Choose'
  1 = 'Tested Terminal'
  2 = 'Reference Terminal'
   = ''
END_TEXTLIST

// ---- VISUs/TextList/TL_Direction.TcTLO
TEXTLIST TL_Direction
  0 = 'Choose'
  1 = 'Input Module'
  2 = 'Output Module'
   = ''
END_TEXTLIST

// ---- VISUs/TextList/TL_Nchannel.TcTLO
TEXTLIST TL_Nchannel
  0 = 'Choose'
  1 = '2 channels'
  2 = '4 channels'
  3 = '8 channels'
   = ''
END_TEXTLIST
